PROGRAM Slit_South
VAR
//Outputs: Power for Limit switches, Home Sensors, etc.
    //bPowerSwitchesAxis1 AT %Q*: BOOL:= TRUE;

//Hardware interlocks
    //bInterlockFwdOK AT %I*: BOOL;
END_VAR

//Initial parameters of an Axis
IF _TaskInfo[fbGetCurTaskIndex.index].FirstCycle THEN
    //Initial default values:
    GVL.astAxes[AXIS_SLIT_SOUTH].stConfig.eHomeSeq := E_HomingRoutines.eHomeToLimit_Fwd;
    GVL.astAxes[AXIS_SLIT_SOUTH].stConfig.fHomePosition := 70.0;
    GVL.astAxes[AXIS_SLIT_SOUTH].stConfig.fHomeFinishDistance := -5.0;
    GVL.astAxes[AXIS_SLIT_SOUTH].stConfig.eRestorePosition := E_RestorePosition.eRestoreWithoutHome;
END_IF

//Define ACTIONS() or write exclusive code for an specific axis.
(*Eg. Stop when temperature reaches certain values, reduce speed if  a signal is activated, etc.
Eg. GVL.astAxes[x].stControl.bInterlockFwd := NOT bInterlockFwdOK;*)
astAxes[AXIS_SLIT_SOUTH].stControl.bEnable:=TRUE;

END_PROGRAM

(* stored: Version 1.1.0.1, ProductVersion 3.1.4024.11
   POU Slit_South: Id {0f1bb328-ea4a-4211-afe7-2cc2c4da3314}, SpecialFunc None *)
